TYPE ST_MGB2IO :
STRUCT
    
END_STRUCT
END_TYPE

(* stored: Version 1.1.0.1, ProductVersion 3.1.4024.12
   DUT ST_MGB2IO: Id {b8e73b8a-6154-489a-9f66-f4ad4eb2cf2f} *)
